{attribute 'qualified_only'}
VAR_GLOBAL
	
	PumpError 	 : ST_PumpError; 
    ValveError 	 : ST_ValveError;
    GeneralAlarm : ST_GeneralAlarm;

END_VAR

(* stored: Version 1.1.0.1, ProductVersion 3.1.4024.12
   GVL GVL_Alarm: Id {6a1f5514-7474-4a0f-8fd8-7c1cd0eaffc0} *)
